// TIA Portal V17 export
// export: Created 2023-03-03T08:59:14.9842508Z, ExportSetting WithDefaults, DisplayName Totally Integrated Automation Portal, DisplayVersion V17 Update 5, DisplayName TIA Portal Openness, DisplayVersion V17 Update 5, DisplayName TIA Portal Version Control Interface, DisplayVersion V17, DisplayName SINAMICS Startdrive Advanced, DisplayVersion V17 SP1, DisplayName SINAMICS DCC, DisplayVersion V17 Update 1, DisplayName SINAMICS Startdrive G130, G150, S120, S150, SINAMICS MV, S210, DisplayVersion V17 SP1, DisplayName SINAMICS Startdrive G110M, G120, G120C, G120D, G120P, G115D, DisplayVersion V17 SP1, DisplayName STEP 7 Professional, DisplayVersion V17 Update 5, DisplayName STEP 7 Safety, DisplayVersion V17, DisplayName WinCC Advanced, DisplayVersion V17 Update 5
FUNCTION "Lubrification" : Void   // FC600, LAD
TITLE = FC Gestione lubrificazione impianto
{ S7_Optimized_Access := 'FALSE' }
AUTHOR : max
FAMILY : Taglio
NAME : FC_LUBRIFICAZIONE
VERSION : 0.1
// stored: AutoNumber false, IsIECCheckEnabled false, SetENOAutomatically false, UDAEnableTagReadback false
   VAR_TEMP   // added for the SCL form of the ladder/FBD networks
      _w1 : Bool;
      _w2 : Bool;
      _w3 : Bool;
      _w4 : Bool;
   END_VAR
BEGIN

REGION Network 1: ****************************** Lubrificazione cesoia *************************************
END_REGION

REGION Network 2: Condizioni per consenso abilitazione
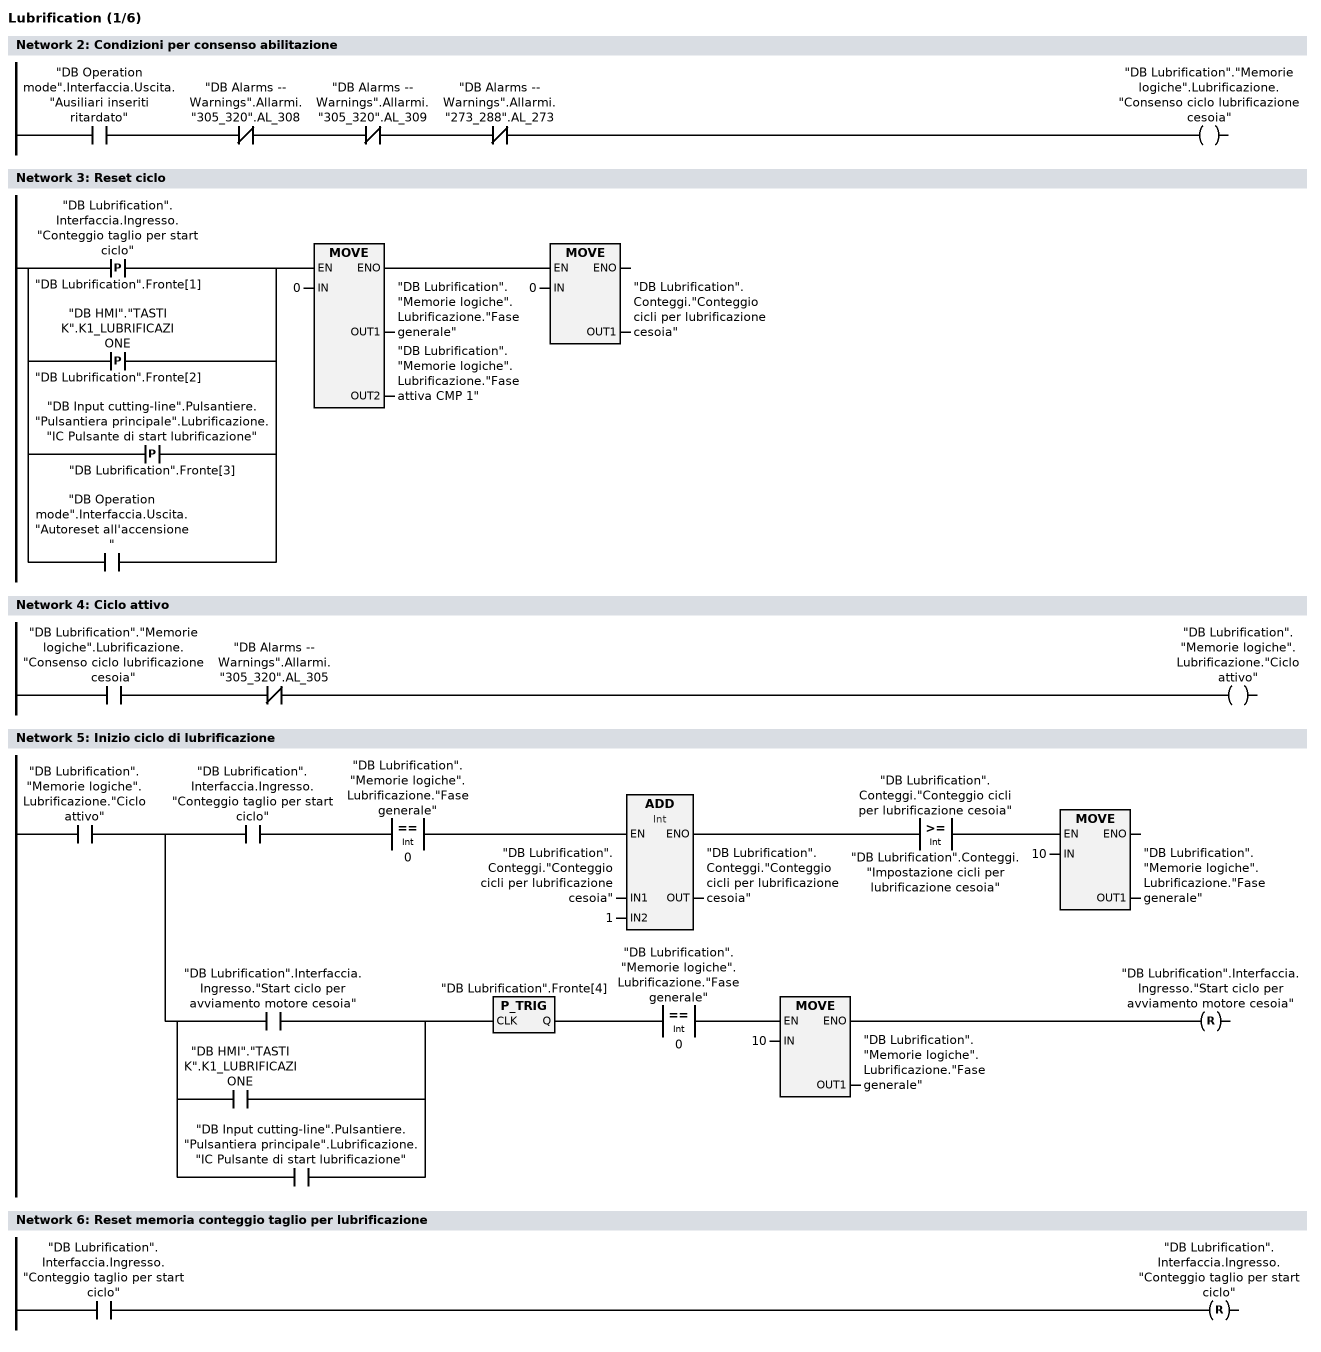
   RUNG wire#powerrail
      Contact( "DB Operation mode".Interfaccia.Uscita."Ausiliari inseriti ritardato" )
      I_Contact( "DB Alarms -- Warnings".Allarmi."305_320".AL_308 )
      I_Contact( "DB Alarms -- Warnings".Allarmi."305_320".AL_309 )
      I_Contact( "DB Alarms -- Warnings".Allarmi."273_288".AL_273 )
      Coil( "DB Lubrification"."Memorie logiche".Lubrificazione."Consenso ciclo lubrificazione cesoia" )
   END_RUNG
   // the same network as SCL:
   "DB Lubrification"."Memorie logiche".Lubrificazione."Consenso ciclo lubrificazione cesoia" := "DB Operation mode".Interfaccia.Uscita."Ausiliari inseriti ritardato" AND NOT "DB Alarms -- Warnings".Allarmi."305_320".AL_308 AND NOT "DB Alarms -- Warnings".Allarmi."305_320".AL_309 AND NOT "DB Alarms -- Warnings".Allarmi."273_288".AL_273;
END_REGION

REGION Network 3: Reset ciclo
   RUNG wire#powerrail
      P_Contact(operand := "DB Lubrification".Interfaccia.Ingresso."Conteggio taglio per start ciclo", bit := "DB Lubrification".Fronte[1])
      wire#w1
      Move(in := 0, out1 => "DB Lubrification"."Memorie logiche".Lubrificazione."Fase generale", out2 => "DB Lubrification"."Memorie logiche".Lubrificazione."Fase attiva CMP 1")
      Move(in := 0, out1 => "DB Lubrification".Conteggi."Conteggio cicli per lubrificazione cesoia")
   END_RUNG
   RUNG wire#powerrail
      P_Contact(operand := "DB HMI"."TASTI K".K1_LUBRIFICAZIONE, bit := "DB Lubrification".Fronte[2])
   END_RUNG wire#w1
   RUNG wire#powerrail
      P_Contact(operand := "DB Input cutting-line".Pulsantiere."Pulsantiera principale".Lubrificazione."IC Pulsante di start lubrificazione", bit := "DB Lubrification".Fronte[3])
   END_RUNG wire#w1
   RUNG wire#powerrail
      Contact( "DB Operation mode".Interfaccia.Uscita."Autoreset all'accensione" )
   END_RUNG wire#w1
   // the same network as SCL:
   #_w1 := "DB Lubrification".Interfaccia.Ingresso."Conteggio taglio per start ciclo" AND NOT "DB Lubrification".Fronte[1];   // rising edge of "DB Lubrification".Interfaccia.Ingresso."Conteggio taglio per start ciclo"
   "DB Lubrification".Fronte[1] := "DB Lubrification".Interfaccia.Ingresso."Conteggio taglio per start ciclo";
   #_w2 := "DB HMI"."TASTI K".K1_LUBRIFICAZIONE AND NOT "DB Lubrification".Fronte[2];   // rising edge of "DB HMI"."TASTI K".K1_LUBRIFICAZIONE
   "DB Lubrification".Fronte[2] := "DB HMI"."TASTI K".K1_LUBRIFICAZIONE;
   #_w3 := "DB Input cutting-line".Pulsantiere."Pulsantiera principale".Lubrificazione."IC Pulsante di start lubrificazione" AND NOT "DB Lubrification".Fronte[3];   // rising edge of "DB Input cutting-line".Pulsantiere."Pulsantiera principale".Lubrificazione."IC Pulsante di start lubrificazione"
   "DB Lubrification".Fronte[3] := "DB Input cutting-line".Pulsantiere."Pulsantiera principale".Lubrificazione."IC Pulsante di start lubrificazione";
   IF #_w1 OR #_w2 OR #_w3 OR "DB Operation mode".Interfaccia.Uscita."Autoreset all'accensione" THEN
       "DB Lubrification"."Memorie logiche".Lubrificazione."Fase generale" := 0;
       "DB Lubrification"."Memorie logiche".Lubrificazione."Fase attiva CMP 1" := 0;
       "DB Lubrification".Conteggi."Conteggio cicli per lubrificazione cesoia" := 0;
   END_IF;
END_REGION

REGION Network 4: Ciclo attivo
   RUNG wire#powerrail
      Contact( "DB Lubrification"."Memorie logiche".Lubrificazione."Consenso ciclo lubrificazione cesoia" )
      I_Contact( "DB Alarms -- Warnings".Allarmi."305_320".AL_305 )
      Coil( "DB Lubrification"."Memorie logiche".Lubrificazione."Ciclo attivo" )
   END_RUNG
   // the same network as SCL:
   "DB Lubrification"."Memorie logiche".Lubrificazione."Ciclo attivo" := "DB Lubrification"."Memorie logiche".Lubrificazione."Consenso ciclo lubrificazione cesoia" AND NOT "DB Alarms -- Warnings".Allarmi."305_320".AL_305;
END_REGION

REGION Network 5: Inizio ciclo di lubrificazione
   RUNG wire#powerrail
      Contact( "DB Lubrification"."Memorie logiche".Lubrificazione."Ciclo attivo" )
      wire#w1
      Contact( "DB Lubrification".Interfaccia.Ingresso."Conteggio taglio per start ciclo" )
      { S7_Templates := "SrcType := Int" } EQ_Contact(in1 := "DB Lubrification"."Memorie logiche".Lubrificazione."Fase generale", in2 := 0)
      { S7_Templates := "SrcType := Int"; S7_GenerateENO := "TRUE" } Add(in1 := "DB Lubrification".Conteggi."Conteggio cicli per lubrificazione cesoia", in2 := 1, out => "DB Lubrification".Conteggi."Conteggio cicli per lubrificazione cesoia")
      { S7_Templates := "SrcType := Int" } GE_Contact(in1 := "DB Lubrification".Conteggi."Conteggio cicli per lubrificazione cesoia", in2 := "DB Lubrification".Conteggi."Impostazione cicli per lubrificazione cesoia")
      Move(in := 10, out1 => "DB Lubrification"."Memorie logiche".Lubrificazione."Fase generale")
   END_RUNG
   RUNG wire#w1
      Contact( "DB Lubrification".Interfaccia.Ingresso."Start ciclo per avviamento motore cesoia" )
      wire#w2
      P_Trig( "DB Lubrification".Fronte[4] )
      { S7_Templates := "SrcType := Int" } EQ_Contact(in1 := "DB Lubrification"."Memorie logiche".Lubrificazione."Fase generale", in2 := 0)
      Move(in := 10, out1 => "DB Lubrification"."Memorie logiche".Lubrificazione."Fase generale")
      R_Coil( "DB Lubrification".Interfaccia.Ingresso."Start ciclo per avviamento motore cesoia" )
   END_RUNG
   RUNG wire#w1
      Contact( "DB HMI"."TASTI K".K1_LUBRIFICAZIONE )
   END_RUNG wire#w2
   RUNG wire#w1
      Contact( "DB Input cutting-line".Pulsantiere."Pulsantiera principale".Lubrificazione."IC Pulsante di start lubrificazione" )
   END_RUNG wire#w2
   // the same network as SCL:
   // ENO of a box is taken as its EN; it also drops when the box reports an error
   #_w1 := "DB Lubrification"."Memorie logiche".Lubrificazione."Ciclo attivo" AND "DB Lubrification".Interfaccia.Ingresso."Conteggio taglio per start ciclo" AND ("DB Lubrification"."Memorie logiche".Lubrificazione."Fase generale" = 0);
   IF #_w1 THEN
       "DB Lubrification".Conteggi."Conteggio cicli per lubrificazione cesoia" := "DB Lubrification".Conteggi."Conteggio cicli per lubrificazione cesoia" + 1;
   END_IF;
   IF #_w1 AND ("DB Lubrification".Conteggi."Conteggio cicli per lubrificazione cesoia" >= "DB Lubrification".Conteggi."Impostazione cicli per lubrificazione cesoia") THEN
       "DB Lubrification"."Memorie logiche".Lubrificazione."Fase generale" := 10;
   END_IF;
   #_w2 := "DB Lubrification"."Memorie logiche".Lubrificazione."Ciclo attivo" AND ("DB Lubrification".Interfaccia.Ingresso."Start ciclo per avviamento motore cesoia" OR "DB HMI"."TASTI K".K1_LUBRIFICAZIONE OR "DB Input cutting-line".Pulsantiere."Pulsantiera principale".Lubrificazione."IC Pulsante di start lubrificazione");
   #_w3 := #_w2 AND NOT "DB Lubrification".Fronte[4];   // rising edge
   "DB Lubrification".Fronte[4] := #_w2;
   #_w4 := #_w3 AND ("DB Lubrification"."Memorie logiche".Lubrificazione."Fase generale" = 0);
   IF #_w4 THEN
       "DB Lubrification"."Memorie logiche".Lubrificazione."Fase generale" := 10;
       "DB Lubrification".Interfaccia.Ingresso."Start ciclo per avviamento motore cesoia" := FALSE;
   END_IF;
END_REGION

REGION Network 6: Reset memoria conteggio taglio per lubrificazione
   RUNG wire#powerrail
      Contact( "DB Lubrification".Interfaccia.Ingresso."Conteggio taglio per start ciclo" )
      R_Coil( "DB Lubrification".Interfaccia.Ingresso."Conteggio taglio per start ciclo" )
   END_RUNG
   // the same network as SCL:
   IF "DB Lubrification".Interfaccia.Ingresso."Conteggio taglio per start ciclo" THEN
       "DB Lubrification".Interfaccia.Ingresso."Conteggio taglio per start ciclo" := FALSE;
   END_IF;
END_REGION

REGION Network 7: Fase10 generale: Verifica stato CMP ad inizio ciclo
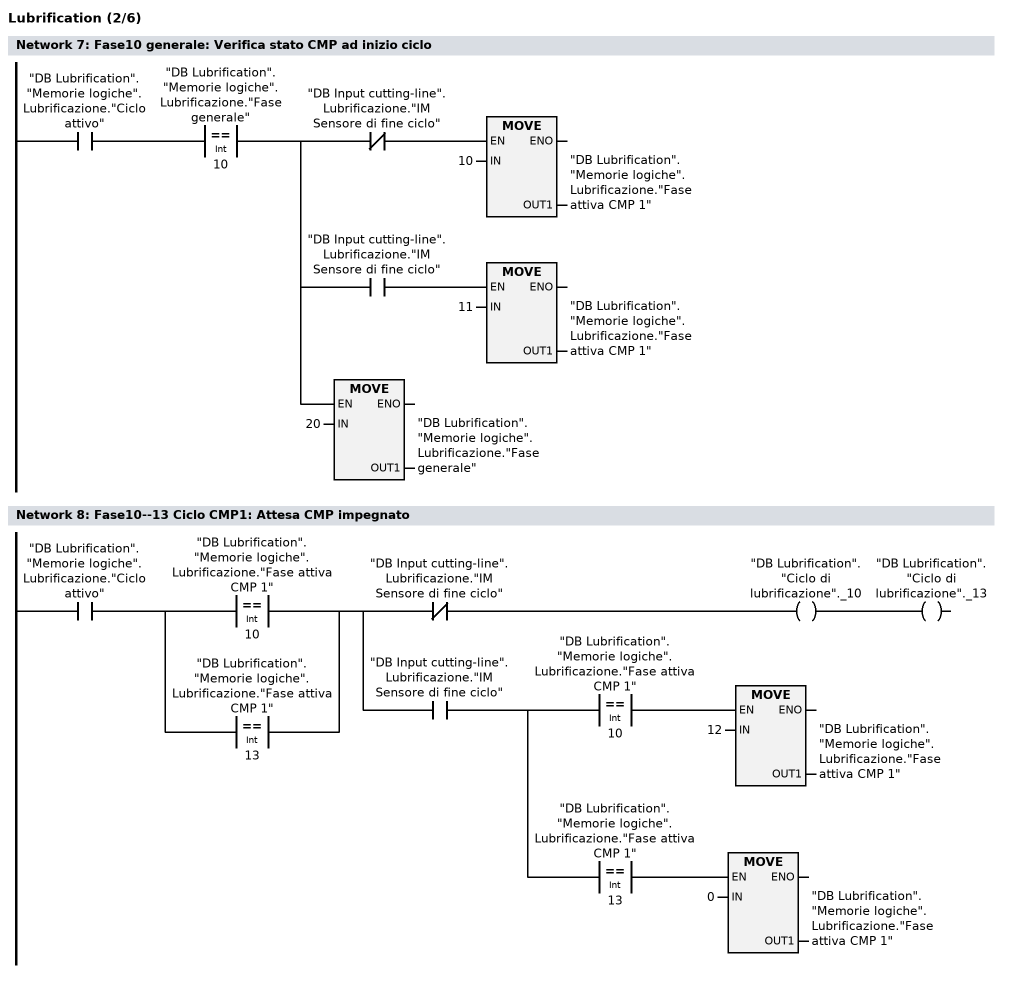
   RUNG wire#powerrail
      Contact( "DB Lubrification"."Memorie logiche".Lubrificazione."Ciclo attivo" )
      { S7_Templates := "SrcType := Int" } EQ_Contact(in1 := "DB Lubrification"."Memorie logiche".Lubrificazione."Fase generale", in2 := 10)
      wire#w1
      I_Contact( "DB Input cutting-line".Lubrificazione."IM Sensore di fine ciclo" )
      Move(in := 10, out1 => "DB Lubrification"."Memorie logiche".Lubrificazione."Fase attiva CMP 1")
   END_RUNG
   RUNG wire#w1
      Contact( "DB Input cutting-line".Lubrificazione."IM Sensore di fine ciclo" )
      Move(in := 11, out1 => "DB Lubrification"."Memorie logiche".Lubrificazione."Fase attiva CMP 1")
   END_RUNG
   RUNG wire#w1
      Move(in := 20, out1 => "DB Lubrification"."Memorie logiche".Lubrificazione."Fase generale")
   END_RUNG
   // the same network as SCL:
   #_w1 := "DB Lubrification"."Memorie logiche".Lubrificazione."Ciclo attivo" AND ("DB Lubrification"."Memorie logiche".Lubrificazione."Fase generale" = 10);
   IF #_w1 AND NOT "DB Input cutting-line".Lubrificazione."IM Sensore di fine ciclo" THEN
       "DB Lubrification"."Memorie logiche".Lubrificazione."Fase attiva CMP 1" := 10;
   END_IF;
   IF #_w1 AND "DB Input cutting-line".Lubrificazione."IM Sensore di fine ciclo" THEN
       "DB Lubrification"."Memorie logiche".Lubrificazione."Fase attiva CMP 1" := 11;
   END_IF;
   IF #_w1 THEN "DB Lubrification"."Memorie logiche".Lubrificazione."Fase generale" := 20; END_IF;
END_REGION

REGION Network 8: Fase10--13 Ciclo CMP1: Attesa CMP impegnato
   RUNG wire#powerrail
      Contact( "DB Lubrification"."Memorie logiche".Lubrificazione."Ciclo attivo" )
      wire#w1
      { S7_Templates := "SrcType := Int" } EQ_Contact(in1 := "DB Lubrification"."Memorie logiche".Lubrificazione."Fase attiva CMP 1", in2 := 10)
      wire#w2
      I_Contact( "DB Input cutting-line".Lubrificazione."IM Sensore di fine ciclo" )
      Coil( "DB Lubrification"."Ciclo di lubrificazione"._10 )
      Coil( "DB Lubrification"."Ciclo di lubrificazione"._13 )
   END_RUNG
   RUNG wire#w1
      { S7_Templates := "SrcType := Int" } EQ_Contact(in1 := "DB Lubrification"."Memorie logiche".Lubrificazione."Fase attiva CMP 1", in2 := 13)
   END_RUNG wire#w2
   RUNG wire#w2
      Contact( "DB Input cutting-line".Lubrificazione."IM Sensore di fine ciclo" )
      wire#w3
      { S7_Templates := "SrcType := Int" } EQ_Contact(in1 := "DB Lubrification"."Memorie logiche".Lubrificazione."Fase attiva CMP 1", in2 := 10)
      Move(in := 12, out1 => "DB Lubrification"."Memorie logiche".Lubrificazione."Fase attiva CMP 1")
   END_RUNG
   RUNG wire#w3
      { S7_Templates := "SrcType := Int" } EQ_Contact(in1 := "DB Lubrification"."Memorie logiche".Lubrificazione."Fase attiva CMP 1", in2 := 13)
      Move(in := 0, out1 => "DB Lubrification"."Memorie logiche".Lubrificazione."Fase attiva CMP 1")
   END_RUNG
   // the same network as SCL:
   #_w1 := "DB Lubrification"."Memorie logiche".Lubrificazione."Ciclo attivo" AND (("DB Lubrification"."Memorie logiche".Lubrificazione."Fase attiva CMP 1" = 10) OR ("DB Lubrification"."Memorie logiche".Lubrificazione."Fase attiva CMP 1" = 13));
   "DB Lubrification"."Ciclo di lubrificazione"._10 := #_w1 AND NOT "DB Input cutting-line".Lubrificazione."IM Sensore di fine ciclo";
   "DB Lubrification"."Ciclo di lubrificazione"._13 := "DB Lubrification"."Ciclo di lubrificazione"._10;
   #_w2 := #_w1 AND "DB Input cutting-line".Lubrificazione."IM Sensore di fine ciclo";
   IF #_w2 AND ("DB Lubrification"."Memorie logiche".Lubrificazione."Fase attiva CMP 1" = 10) THEN
       "DB Lubrification"."Memorie logiche".Lubrificazione."Fase attiva CMP 1" := 12;
   END_IF;
   IF #_w2 AND ("DB Lubrification"."Memorie logiche".Lubrificazione."Fase attiva CMP 1" = 13) THEN
       "DB Lubrification"."Memorie logiche".Lubrificazione."Fase attiva CMP 1" := 0;
   END_IF;
END_REGION

REGION Network 9: Fase11--12 Ciclo CMP1: Attesa CMP dimpegnato
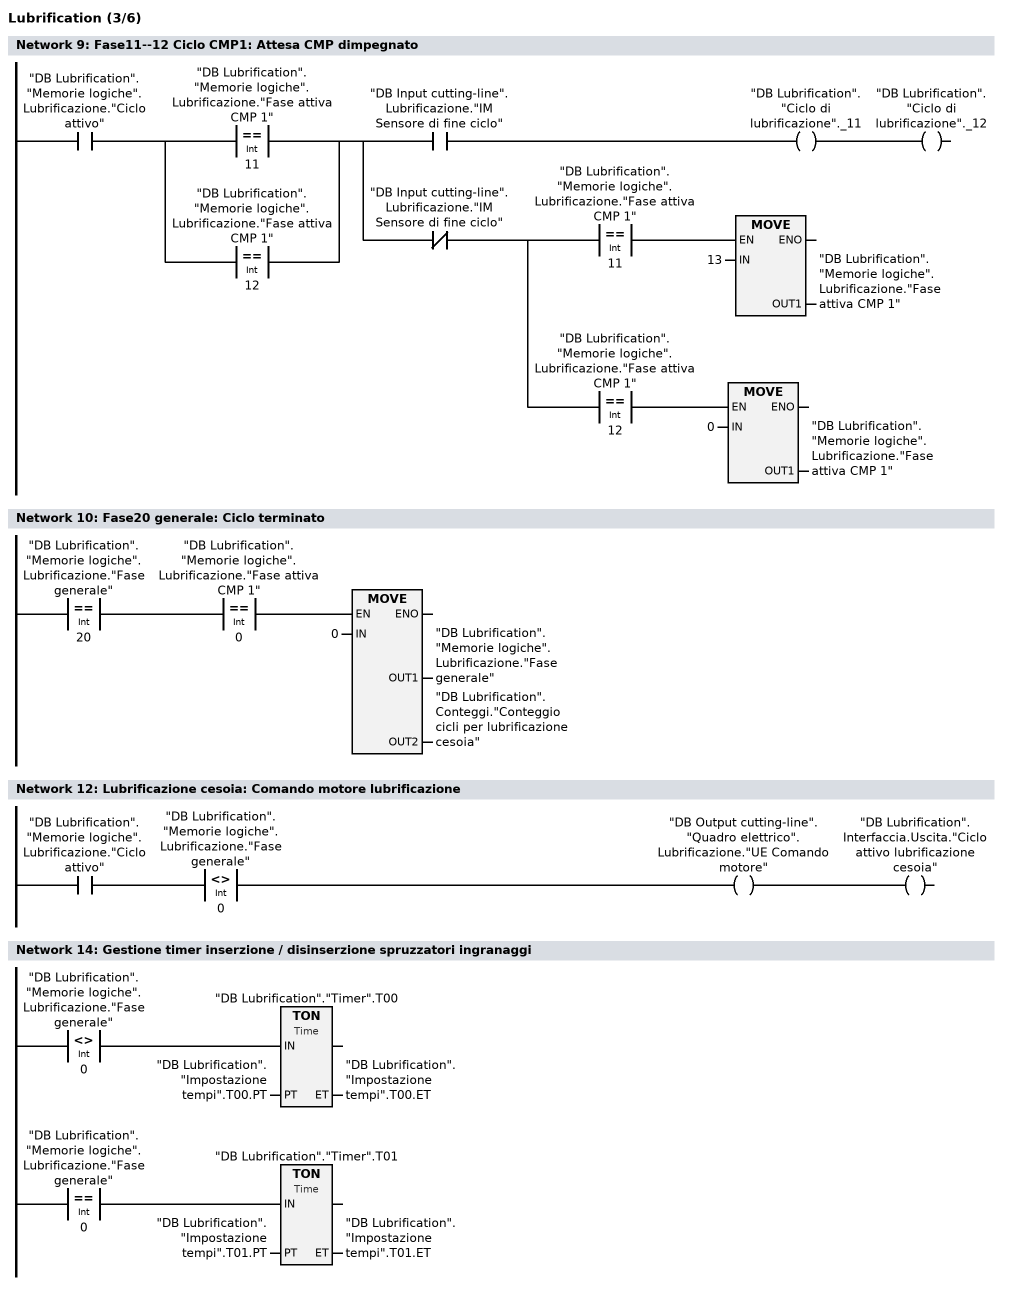
   RUNG wire#powerrail
      Contact( "DB Lubrification"."Memorie logiche".Lubrificazione."Ciclo attivo" )
      wire#w1
      { S7_Templates := "SrcType := Int" } EQ_Contact(in1 := "DB Lubrification"."Memorie logiche".Lubrificazione."Fase attiva CMP 1", in2 := 11)
      wire#w2
      Contact( "DB Input cutting-line".Lubrificazione."IM Sensore di fine ciclo" )
      Coil( "DB Lubrification"."Ciclo di lubrificazione"._11 )
      Coil( "DB Lubrification"."Ciclo di lubrificazione"._12 )
   END_RUNG
   RUNG wire#w1
      { S7_Templates := "SrcType := Int" } EQ_Contact(in1 := "DB Lubrification"."Memorie logiche".Lubrificazione."Fase attiva CMP 1", in2 := 12)
   END_RUNG wire#w2
   RUNG wire#w2
      I_Contact( "DB Input cutting-line".Lubrificazione."IM Sensore di fine ciclo" )
      wire#w3
      { S7_Templates := "SrcType := Int" } EQ_Contact(in1 := "DB Lubrification"."Memorie logiche".Lubrificazione."Fase attiva CMP 1", in2 := 11)
      Move(in := 13, out1 => "DB Lubrification"."Memorie logiche".Lubrificazione."Fase attiva CMP 1")
   END_RUNG
   RUNG wire#w3
      { S7_Templates := "SrcType := Int" } EQ_Contact(in1 := "DB Lubrification"."Memorie logiche".Lubrificazione."Fase attiva CMP 1", in2 := 12)
      Move(in := 0, out1 => "DB Lubrification"."Memorie logiche".Lubrificazione."Fase attiva CMP 1")
   END_RUNG
   // the same network as SCL:
   #_w1 := "DB Lubrification"."Memorie logiche".Lubrificazione."Ciclo attivo" AND (("DB Lubrification"."Memorie logiche".Lubrificazione."Fase attiva CMP 1" = 11) OR ("DB Lubrification"."Memorie logiche".Lubrificazione."Fase attiva CMP 1" = 12));
   "DB Lubrification"."Ciclo di lubrificazione"._11 := #_w1 AND "DB Input cutting-line".Lubrificazione."IM Sensore di fine ciclo";
   "DB Lubrification"."Ciclo di lubrificazione"._12 := "DB Lubrification"."Ciclo di lubrificazione"._11;
   #_w2 := #_w1 AND NOT "DB Input cutting-line".Lubrificazione."IM Sensore di fine ciclo";
   IF #_w2 AND ("DB Lubrification"."Memorie logiche".Lubrificazione."Fase attiva CMP 1" = 11) THEN
       "DB Lubrification"."Memorie logiche".Lubrificazione."Fase attiva CMP 1" := 13;
   END_IF;
   IF #_w2 AND ("DB Lubrification"."Memorie logiche".Lubrificazione."Fase attiva CMP 1" = 12) THEN
       "DB Lubrification"."Memorie logiche".Lubrificazione."Fase attiva CMP 1" := 0;
   END_IF;
END_REGION

REGION Network 10: Fase20 generale: Ciclo terminato
   RUNG wire#powerrail
      { S7_Templates := "SrcType := Int" } EQ_Contact(in1 := "DB Lubrification"."Memorie logiche".Lubrificazione."Fase generale", in2 := 20)
      { S7_Templates := "SrcType := Int" } EQ_Contact(in1 := "DB Lubrification"."Memorie logiche".Lubrificazione."Fase attiva CMP 1", in2 := 0)
      Move(in := 0, out1 => "DB Lubrification"."Memorie logiche".Lubrificazione."Fase generale", out2 => "DB Lubrification".Conteggi."Conteggio cicli per lubrificazione cesoia")
   END_RUNG
   // the same network as SCL:
   IF ("DB Lubrification"."Memorie logiche".Lubrificazione."Fase generale" = 20) AND ("DB Lubrification"."Memorie logiche".Lubrificazione."Fase attiva CMP 1" = 0) THEN
       "DB Lubrification"."Memorie logiche".Lubrificazione."Fase generale" := 0;
       "DB Lubrification".Conteggi."Conteggio cicli per lubrificazione cesoia" := 0;
   END_IF;
END_REGION

REGION Network 11: Dummy
END_REGION

REGION Network 12: Lubrificazione cesoia: Comando motore lubrificazione
   RUNG wire#powerrail
      Contact( "DB Lubrification"."Memorie logiche".Lubrificazione."Ciclo attivo" )
      { S7_Templates := "SrcType := Int" } NE_Contact(in1 := "DB Lubrification"."Memorie logiche".Lubrificazione."Fase generale", in2 := 0)
      Coil( "DB Output cutting-line"."Quadro elettrico".Lubrificazione."UE Comando motore" )
      Coil( "DB Lubrification".Interfaccia.Uscita."Ciclo attivo lubrificazione cesoia" )
   END_RUNG
   // the same network as SCL:
   "DB Output cutting-line"."Quadro elettrico".Lubrificazione."UE Comando motore" := "DB Lubrification"."Memorie logiche".Lubrificazione."Ciclo attivo" AND ("DB Lubrification"."Memorie logiche".Lubrificazione."Fase generale" <> 0);
   "DB Lubrification".Interfaccia.Uscita."Ciclo attivo lubrificazione cesoia" := "DB Output cutting-line"."Quadro elettrico".Lubrificazione."UE Comando motore";
END_REGION

REGION Network 13: Dummy
END_REGION

REGION Network 14: Gestione timer inserzione / disinserzione spruzzatori ingranaggi
   RUNG wire#powerrail
      { S7_Templates := "SrcType := Int" } NE_Contact(in1 := "DB Lubrification"."Memorie logiche".Lubrificazione."Fase generale", in2 := 0)
      { S7_Templates := "time_type := Time" } "DB Lubrification"."Timer".T00.TON(pt := "DB Lubrification"."Impostazione tempi".T00.PT, et => "DB Lubrification"."Impostazione tempi".T00.ET)
   END_RUNG
   RUNG wire#powerrail
      { S7_Templates := "SrcType := Int" } EQ_Contact(in1 := "DB Lubrification"."Memorie logiche".Lubrificazione."Fase generale", in2 := 0)
      { S7_Templates := "time_type := Time" } "DB Lubrification"."Timer".T01.TON(pt := "DB Lubrification"."Impostazione tempi".T01.PT, et => "DB Lubrification"."Impostazione tempi".T01.ET)
   END_RUNG
   // the same network as SCL:
   "DB Lubrification"."Timer".T00.TON(IN := "DB Lubrification"."Memorie logiche".Lubrificazione."Fase generale" <> 0,
                           PT := "DB Lubrification"."Impostazione tempi".T00.PT,
                           ET => "DB Lubrification"."Impostazione tempi".T00.ET);
   "DB Lubrification"."Timer".T01.TON(IN := "DB Lubrification"."Memorie logiche".Lubrificazione."Fase generale" = 0,
                           PT := "DB Lubrification"."Impostazione tempi".T01.PT,
                           ET => "DB Lubrification"."Impostazione tempi".T01.ET);
END_REGION

REGION Network 15: Lubrificazione cesoia: Comando spruzzatori ingranaggi
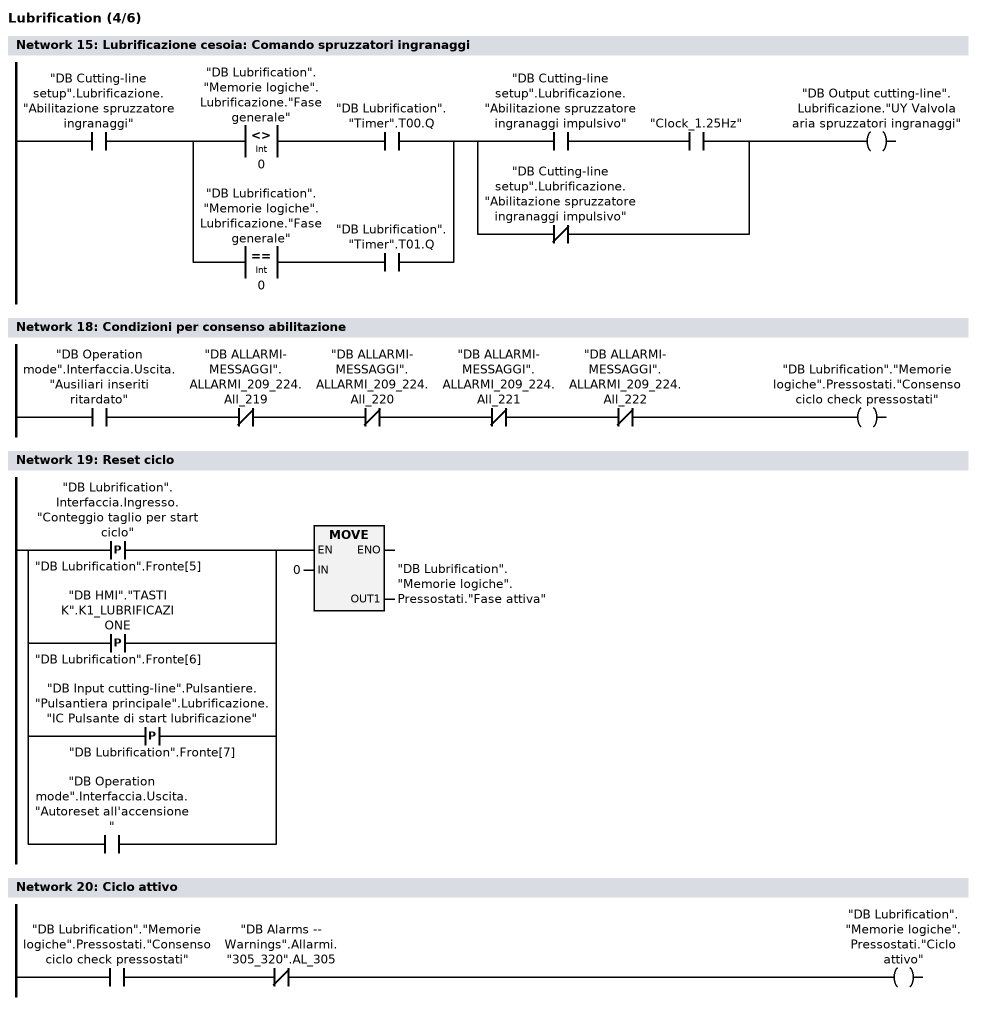
   RUNG wire#powerrail
      Contact( "DB Cutting-line setup".Lubrificazione."Abilitazione spruzzatore ingranaggi" )
      wire#w1
      { S7_Templates := "SrcType := Int" } NE_Contact(in1 := "DB Lubrification"."Memorie logiche".Lubrificazione."Fase generale", in2 := 0)
      Contact( "DB Lubrification"."Timer".T00.Q )
      wire#w2
      Contact( "DB Cutting-line setup".Lubrificazione."Abilitazione spruzzatore ingranaggi impulsivo" )
      Contact( "Clock_1.25Hz" )
      wire#w3
      Coil( "DB Output cutting-line".Lubrificazione."UY Valvola aria spruzzatori ingranaggi" )
   END_RUNG
   RUNG wire#w1
      { S7_Templates := "SrcType := Int" } EQ_Contact(in1 := "DB Lubrification"."Memorie logiche".Lubrificazione."Fase generale", in2 := 0)
      Contact( "DB Lubrification"."Timer".T01.Q )
   END_RUNG wire#w2
   RUNG wire#w2
      I_Contact( "DB Cutting-line setup".Lubrificazione."Abilitazione spruzzatore ingranaggi impulsivo" )
   END_RUNG wire#w3
   // the same network as SCL:
   "DB Output cutting-line".Lubrificazione."UY Valvola aria spruzzatori ingranaggi" := "DB Cutting-line setup".Lubrificazione."Abilitazione spruzzatore ingranaggi" AND ((("DB Lubrification"."Memorie logiche".Lubrificazione."Fase generale" <> 0) AND "DB Lubrification"."Timer".T00.Q) OR (("DB Lubrification"."Memorie logiche".Lubrificazione."Fase generale" = 0) AND "DB Lubrification"."Timer".T01.Q)) AND (("DB Cutting-line setup".Lubrificazione."Abilitazione spruzzatore ingranaggi impulsivo" AND "Clock_1.25Hz") OR NOT "DB Cutting-line setup".Lubrificazione."Abilitazione spruzzatore ingranaggi impulsivo");
END_REGION

REGION Network 16: Dummy
END_REGION

REGION Network 17: ******************************* Check pressostati **************************************
END_REGION

REGION Network 18: Condizioni per consenso abilitazione
   RUNG wire#powerrail
      Contact( "DB Operation mode".Interfaccia.Uscita."Ausiliari inseriti ritardato" )
      I_Contact( "DB ALLARMI-MESSAGGI".ALLARMI_209_224.All_219 )
      I_Contact( "DB ALLARMI-MESSAGGI".ALLARMI_209_224.All_220 )
      I_Contact( "DB ALLARMI-MESSAGGI".ALLARMI_209_224.All_221 )
      I_Contact( "DB ALLARMI-MESSAGGI".ALLARMI_209_224.All_222 )
      Coil( "DB Lubrification"."Memorie logiche".Pressostati."Consenso ciclo check pressostati" )
   END_RUNG
   // the same network as SCL:
   "DB Lubrification"."Memorie logiche".Pressostati."Consenso ciclo check pressostati" := "DB Operation mode".Interfaccia.Uscita."Ausiliari inseriti ritardato" AND NOT "DB ALLARMI-MESSAGGI".ALLARMI_209_224.All_219 AND NOT "DB ALLARMI-MESSAGGI".ALLARMI_209_224.All_220 AND NOT "DB ALLARMI-MESSAGGI".ALLARMI_209_224.All_221 AND NOT "DB ALLARMI-MESSAGGI".ALLARMI_209_224.All_222;
END_REGION

REGION Network 19: Reset ciclo
   RUNG wire#powerrail
      P_Contact(operand := "DB Lubrification".Interfaccia.Ingresso."Conteggio taglio per start ciclo", bit := "DB Lubrification".Fronte[5])
      wire#w1
      Move(in := 0, out1 => "DB Lubrification"."Memorie logiche".Pressostati."Fase attiva")
   END_RUNG
   RUNG wire#powerrail
      P_Contact(operand := "DB HMI"."TASTI K".K1_LUBRIFICAZIONE, bit := "DB Lubrification".Fronte[6])
   END_RUNG wire#w1
   RUNG wire#powerrail
      P_Contact(operand := "DB Input cutting-line".Pulsantiere."Pulsantiera principale".Lubrificazione."IC Pulsante di start lubrificazione", bit := "DB Lubrification".Fronte[7])
   END_RUNG wire#w1
   RUNG wire#powerrail
      Contact( "DB Operation mode".Interfaccia.Uscita."Autoreset all'accensione" )
   END_RUNG wire#w1
   // the same network as SCL:
   #_w1 := "DB Lubrification".Interfaccia.Ingresso."Conteggio taglio per start ciclo" AND NOT "DB Lubrification".Fronte[5];   // rising edge of "DB Lubrification".Interfaccia.Ingresso."Conteggio taglio per start ciclo"
   "DB Lubrification".Fronte[5] := "DB Lubrification".Interfaccia.Ingresso."Conteggio taglio per start ciclo";
   #_w2 := "DB HMI"."TASTI K".K1_LUBRIFICAZIONE AND NOT "DB Lubrification".Fronte[6];   // rising edge of "DB HMI"."TASTI K".K1_LUBRIFICAZIONE
   "DB Lubrification".Fronte[6] := "DB HMI"."TASTI K".K1_LUBRIFICAZIONE;
   #_w3 := "DB Input cutting-line".Pulsantiere."Pulsantiera principale".Lubrificazione."IC Pulsante di start lubrificazione" AND NOT "DB Lubrification".Fronte[7];   // rising edge of "DB Input cutting-line".Pulsantiere."Pulsantiera principale".Lubrificazione."IC Pulsante di start lubrificazione"
   "DB Lubrification".Fronte[7] := "DB Input cutting-line".Pulsantiere."Pulsantiera principale".Lubrificazione."IC Pulsante di start lubrificazione";
   IF #_w1 OR #_w2 OR #_w3 OR "DB Operation mode".Interfaccia.Uscita."Autoreset all'accensione" THEN
       "DB Lubrification"."Memorie logiche".Pressostati."Fase attiva" := 0;
   END_IF;
END_REGION

REGION Network 20: Ciclo attivo
   RUNG wire#powerrail
      Contact( "DB Lubrification"."Memorie logiche".Pressostati."Consenso ciclo check pressostati" )
      I_Contact( "DB Alarms -- Warnings".Allarmi."305_320".AL_305 )
      Coil( "DB Lubrification"."Memorie logiche".Pressostati."Ciclo attivo" )
   END_RUNG
   // the same network as SCL:
   "DB Lubrification"."Memorie logiche".Pressostati."Ciclo attivo" := "DB Lubrification"."Memorie logiche".Pressostati."Consenso ciclo check pressostati" AND NOT "DB Alarms -- Warnings".Allarmi."305_320".AL_305;
END_REGION

REGION Network 21: Inizio ciclo check pressostati
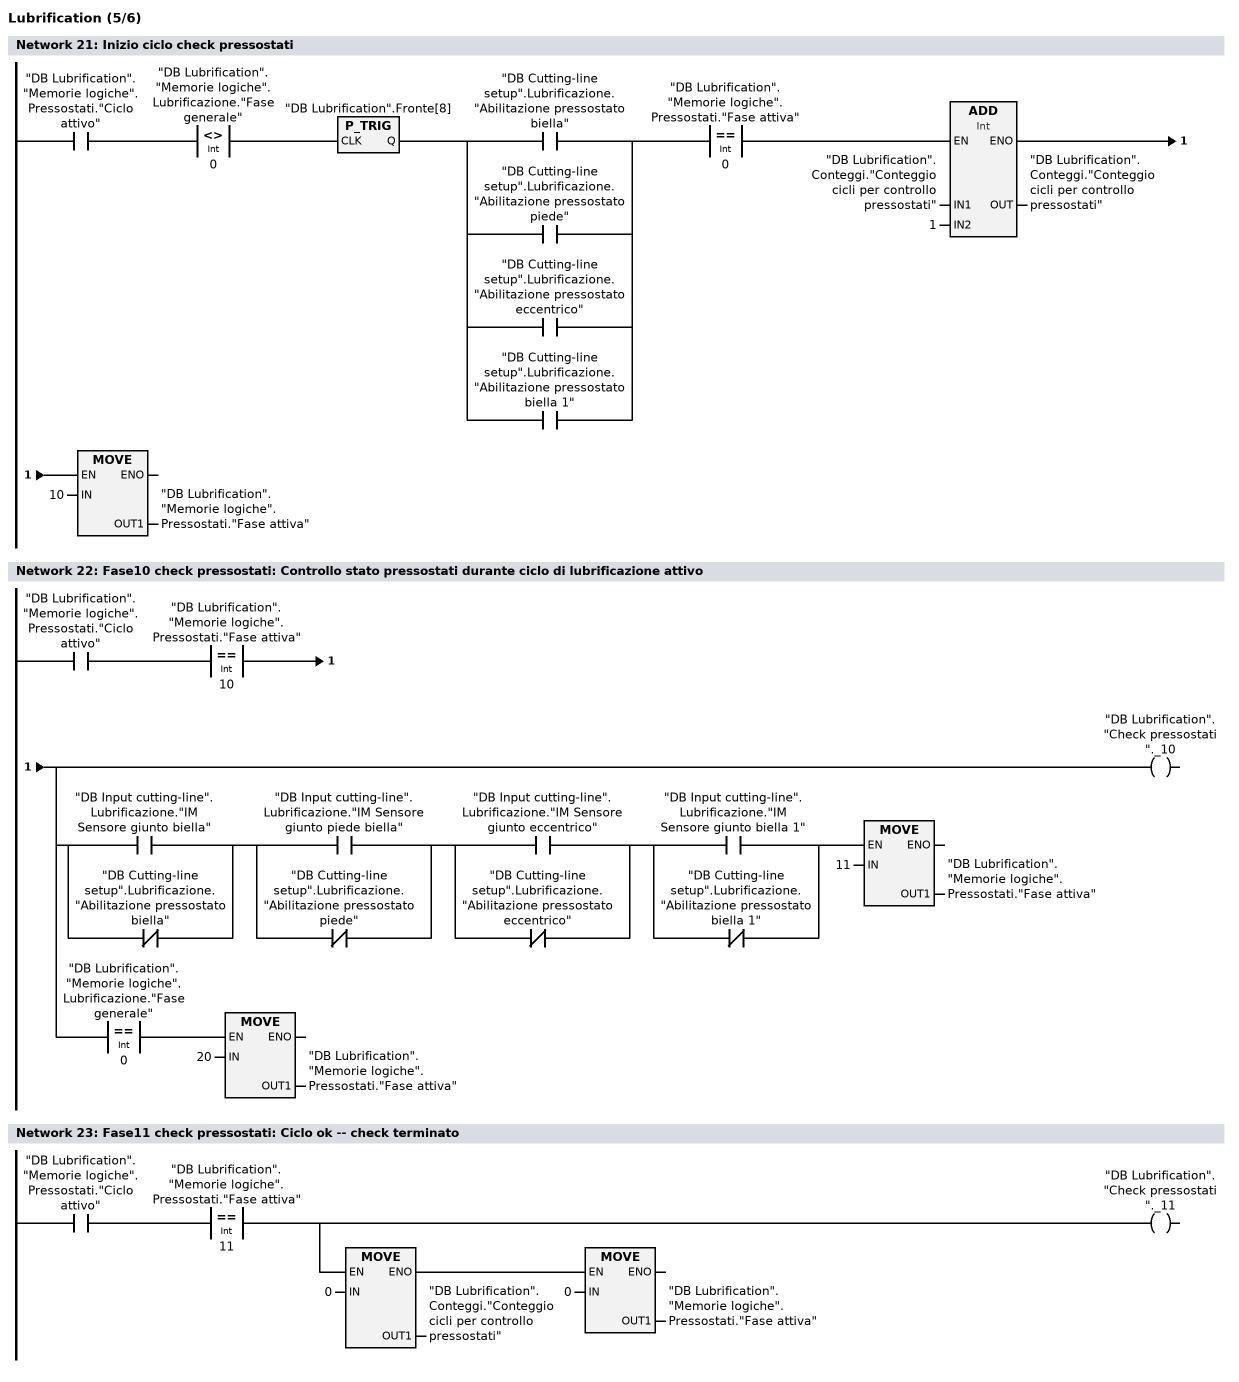
   RUNG wire#powerrail
      Contact( "DB Lubrification"."Memorie logiche".Pressostati."Ciclo attivo" )
      { S7_Templates := "SrcType := Int" } NE_Contact(in1 := "DB Lubrification"."Memorie logiche".Lubrificazione."Fase generale", in2 := 0)
      P_Trig( "DB Lubrification".Fronte[8] )
      wire#w1
      Contact( "DB Cutting-line setup".Lubrificazione."Abilitazione pressostato biella" )
      wire#w2
      { S7_Templates := "SrcType := Int" } EQ_Contact(in1 := "DB Lubrification"."Memorie logiche".Pressostati."Fase attiva", in2 := 0)
      { S7_Templates := "SrcType := Int"; S7_GenerateENO := "TRUE" } Add(in1 := "DB Lubrification".Conteggi."Conteggio cicli per controllo pressostati", in2 := 1, out => "DB Lubrification".Conteggi."Conteggio cicli per controllo pressostati")
      Move(in := 10, out1 => "DB Lubrification"."Memorie logiche".Pressostati."Fase attiva")
   END_RUNG
   RUNG wire#w1
      Contact( "DB Cutting-line setup".Lubrificazione."Abilitazione pressostato piede" )
   END_RUNG wire#w2
   RUNG wire#w1
      Contact( "DB Cutting-line setup".Lubrificazione."Abilitazione pressostato eccentrico" )
   END_RUNG wire#w2
   RUNG wire#w1
      Contact( "DB Cutting-line setup".Lubrificazione."Abilitazione pressostato biella 1" )
   END_RUNG wire#w2
   // the same network as SCL:
   // ENO of a box is taken as its EN; it also drops when the box reports an error
   #_w1 := "DB Lubrification"."Memorie logiche".Pressostati."Ciclo attivo" AND ("DB Lubrification"."Memorie logiche".Lubrificazione."Fase generale" <> 0);
   #_w2 := #_w1 AND NOT "DB Lubrification".Fronte[8];   // rising edge
   "DB Lubrification".Fronte[8] := #_w1;
   IF #_w2 AND ("DB Cutting-line setup".Lubrificazione."Abilitazione pressostato biella" OR "DB Cutting-line setup".Lubrificazione."Abilitazione pressostato piede" OR "DB Cutting-line setup".Lubrificazione."Abilitazione pressostato eccentrico" OR "DB Cutting-line setup".Lubrificazione."Abilitazione pressostato biella 1") AND ("DB Lubrification"."Memorie logiche".Pressostati."Fase attiva" = 0) THEN
       "DB Lubrification".Conteggi."Conteggio cicli per controllo pressostati" := "DB Lubrification".Conteggi."Conteggio cicli per controllo pressostati" + 1;
       "DB Lubrification"."Memorie logiche".Pressostati."Fase attiva" := 10;
   END_IF;
END_REGION

REGION Network 22: Fase10 check pressostati: Controllo stato pressostati durante ciclo di lubrificazione attivo
   RUNG wire#powerrail
      Contact( "DB Lubrification"."Memorie logiche".Pressostati."Ciclo attivo" )
      { S7_Templates := "SrcType := Int" } EQ_Contact(in1 := "DB Lubrification"."Memorie logiche".Pressostati."Fase attiva", in2 := 10)
      wire#w1
      Coil( "DB Lubrification"."Check pressostati"._10 )
   END_RUNG
   RUNG wire#w1
      Contact( "DB Input cutting-line".Lubrificazione."IM Sensore giunto biella" )
      wire#w2
      Contact( "DB Input cutting-line".Lubrificazione."IM Sensore giunto piede biella" )
      wire#w3
      Contact( "DB Input cutting-line".Lubrificazione."IM Sensore giunto eccentrico" )
      wire#w4
      Contact( "DB Input cutting-line".Lubrificazione."IM Sensore giunto biella 1" )
      wire#w5
      Move(in := 11, out1 => "DB Lubrification"."Memorie logiche".Pressostati."Fase attiva")
   END_RUNG
   RUNG wire#w1
      I_Contact( "DB Cutting-line setup".Lubrificazione."Abilitazione pressostato biella" )
   END_RUNG wire#w2
   RUNG wire#w2
      I_Contact( "DB Cutting-line setup".Lubrificazione."Abilitazione pressostato piede" )
   END_RUNG wire#w3
   RUNG wire#w3
      I_Contact( "DB Cutting-line setup".Lubrificazione."Abilitazione pressostato eccentrico" )
   END_RUNG wire#w4
   RUNG wire#w4
      I_Contact( "DB Cutting-line setup".Lubrificazione."Abilitazione pressostato biella 1" )
   END_RUNG wire#w5
   RUNG wire#w1
      { S7_Templates := "SrcType := Int" } EQ_Contact(in1 := "DB Lubrification"."Memorie logiche".Lubrificazione."Fase generale", in2 := 0)
      Move(in := 20, out1 => "DB Lubrification"."Memorie logiche".Pressostati."Fase attiva")
   END_RUNG
   // the same network as SCL:
   "DB Lubrification"."Check pressostati"._10 := "DB Lubrification"."Memorie logiche".Pressostati."Ciclo attivo" AND ("DB Lubrification"."Memorie logiche".Pressostati."Fase attiva" = 10);
   IF "DB Lubrification"."Check pressostati"._10 AND ("DB Input cutting-line".Lubrificazione."IM Sensore giunto biella" OR NOT "DB Cutting-line setup".Lubrificazione."Abilitazione pressostato biella") AND ("DB Input cutting-line".Lubrificazione."IM Sensore giunto piede biella" OR NOT "DB Cutting-line setup".Lubrificazione."Abilitazione pressostato piede") AND ("DB Input cutting-line".Lubrificazione."IM Sensore giunto eccentrico" OR NOT "DB Cutting-line setup".Lubrificazione."Abilitazione pressostato eccentrico") AND ("DB Input cutting-line".Lubrificazione."IM Sensore giunto biella 1" OR NOT "DB Cutting-line setup".Lubrificazione."Abilitazione pressostato biella 1") THEN
       "DB Lubrification"."Memorie logiche".Pressostati."Fase attiva" := 11;
   END_IF;
   IF "DB Lubrification"."Check pressostati"._10 AND ("DB Lubrification"."Memorie logiche".Lubrificazione."Fase generale" = 0) THEN
       "DB Lubrification"."Memorie logiche".Pressostati."Fase attiva" := 20;
   END_IF;
END_REGION

REGION Network 23: Fase11 check pressostati: Ciclo ok -- check terminato
   RUNG wire#powerrail
      Contact( "DB Lubrification"."Memorie logiche".Pressostati."Ciclo attivo" )
      { S7_Templates := "SrcType := Int" } EQ_Contact(in1 := "DB Lubrification"."Memorie logiche".Pressostati."Fase attiva", in2 := 11)
      wire#w1
      Coil( "DB Lubrification"."Check pressostati"._11 )
   END_RUNG
   RUNG wire#w1
      { S7_GenerateENO := "TRUE" } Move(in := 0, out1 => "DB Lubrification".Conteggi."Conteggio cicli per controllo pressostati")
      Move(in := 0, out1 => "DB Lubrification"."Memorie logiche".Pressostati."Fase attiva")
   END_RUNG
   // the same network as SCL:
   // ENO of a box is taken as its EN; it also drops when the box reports an error
   "DB Lubrification"."Check pressostati"._11 := "DB Lubrification"."Memorie logiche".Pressostati."Ciclo attivo" AND ("DB Lubrification"."Memorie logiche".Pressostati."Fase attiva" = 11);
   IF "DB Lubrification"."Check pressostati"._11 THEN
       "DB Lubrification".Conteggi."Conteggio cicli per controllo pressostati" := 0;
       "DB Lubrification"."Memorie logiche".Pressostati."Fase attiva" := 0;
   END_IF;
END_REGION

REGION Network 24: Fase20 check pressostati: Ciclo non ok -- generazione allarmi pressostati se conteggio terminato
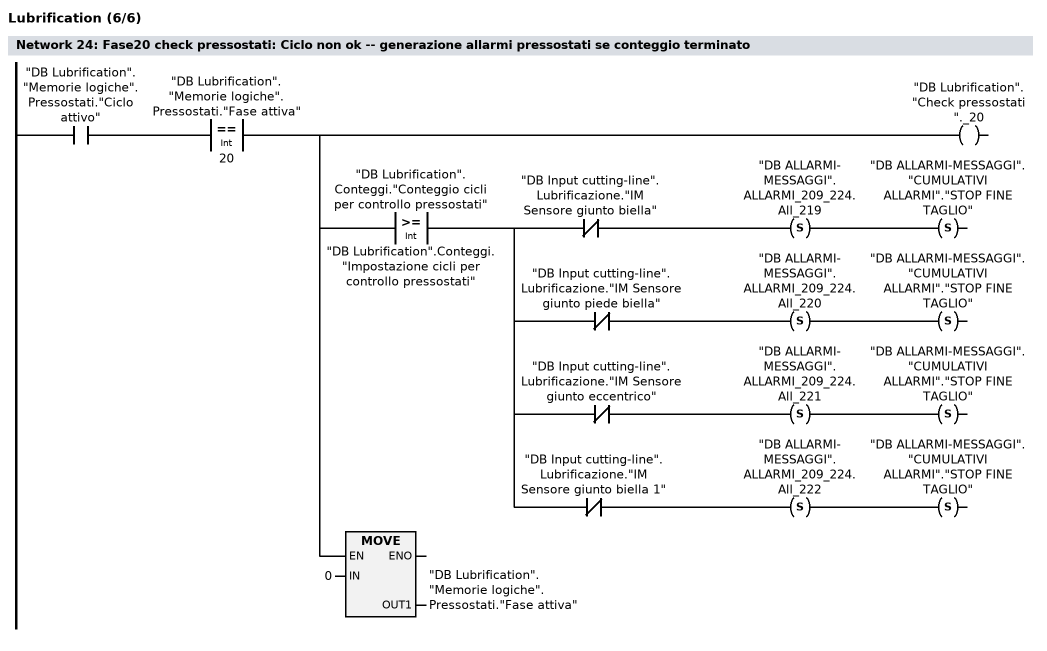
   RUNG wire#powerrail
      Contact( "DB Lubrification"."Memorie logiche".Pressostati."Ciclo attivo" )
      { S7_Templates := "SrcType := Int" } EQ_Contact(in1 := "DB Lubrification"."Memorie logiche".Pressostati."Fase attiva", in2 := 20)
      wire#w1
      Coil( "DB Lubrification"."Check pressostati"._20 )
   END_RUNG
   RUNG wire#w1
      { S7_Templates := "SrcType := Int" } GE_Contact(in1 := "DB Lubrification".Conteggi."Conteggio cicli per controllo pressostati", in2 := "DB Lubrification".Conteggi."Impostazione cicli per controllo pressostati")
      wire#w2
      I_Contact( "DB Input cutting-line".Lubrificazione."IM Sensore giunto biella" )
      S_Coil( "DB ALLARMI-MESSAGGI".ALLARMI_209_224.All_219 )
      S_Coil( "DB ALLARMI-MESSAGGI"."CUMULATIVI ALLARMI"."STOP FINE TAGLIO" )
   END_RUNG
   RUNG wire#w2
      I_Contact( "DB Input cutting-line".Lubrificazione."IM Sensore giunto piede biella" )
      S_Coil( "DB ALLARMI-MESSAGGI".ALLARMI_209_224.All_220 )
      S_Coil( "DB ALLARMI-MESSAGGI"."CUMULATIVI ALLARMI"."STOP FINE TAGLIO" )
   END_RUNG
   RUNG wire#w2
      I_Contact( "DB Input cutting-line".Lubrificazione."IM Sensore giunto eccentrico" )
      S_Coil( "DB ALLARMI-MESSAGGI".ALLARMI_209_224.All_221 )
      S_Coil( "DB ALLARMI-MESSAGGI"."CUMULATIVI ALLARMI"."STOP FINE TAGLIO" )
   END_RUNG
   RUNG wire#w2
      I_Contact( "DB Input cutting-line".Lubrificazione."IM Sensore giunto biella 1" )
      S_Coil( "DB ALLARMI-MESSAGGI".ALLARMI_209_224.All_222 )
      S_Coil( "DB ALLARMI-MESSAGGI"."CUMULATIVI ALLARMI"."STOP FINE TAGLIO" )
   END_RUNG
   RUNG wire#w1
      Move(in := 0, out1 => "DB Lubrification"."Memorie logiche".Pressostati."Fase attiva")
   END_RUNG
   // the same network as SCL:
   "DB Lubrification"."Check pressostati"._20 := "DB Lubrification"."Memorie logiche".Pressostati."Ciclo attivo" AND ("DB Lubrification"."Memorie logiche".Pressostati."Fase attiva" = 20);
   #_w1 := "DB Lubrification"."Check pressostati"._20 AND ("DB Lubrification".Conteggi."Conteggio cicli per controllo pressostati" >= "DB Lubrification".Conteggi."Impostazione cicli per controllo pressostati");
   IF #_w1 AND NOT "DB Input cutting-line".Lubrificazione."IM Sensore giunto biella" THEN
       "DB ALLARMI-MESSAGGI".ALLARMI_209_224.All_219 := TRUE;
       "DB ALLARMI-MESSAGGI"."CUMULATIVI ALLARMI"."STOP FINE TAGLIO" := TRUE;
   END_IF;
   IF #_w1 AND NOT "DB Input cutting-line".Lubrificazione."IM Sensore giunto piede biella" THEN
       "DB ALLARMI-MESSAGGI".ALLARMI_209_224.All_220 := TRUE;
       "DB ALLARMI-MESSAGGI"."CUMULATIVI ALLARMI"."STOP FINE TAGLIO" := TRUE;
   END_IF;
   IF #_w1 AND NOT "DB Input cutting-line".Lubrificazione."IM Sensore giunto eccentrico" THEN
       "DB ALLARMI-MESSAGGI".ALLARMI_209_224.All_221 := TRUE;
       "DB ALLARMI-MESSAGGI"."CUMULATIVI ALLARMI"."STOP FINE TAGLIO" := TRUE;
   END_IF;
   IF #_w1 AND NOT "DB Input cutting-line".Lubrificazione."IM Sensore giunto biella 1" THEN
       "DB ALLARMI-MESSAGGI".ALLARMI_209_224.All_222 := TRUE;
       "DB ALLARMI-MESSAGGI"."CUMULATIVI ALLARMI"."STOP FINE TAGLIO" := TRUE;
   END_IF;
   IF "DB Lubrification"."Check pressostati"._20 THEN
       "DB Lubrification"."Memorie logiche".Pressostati."Fase attiva" := 0;
   END_IF;
END_REGION

REGION Network 25: Dummy
END_REGION
END_FUNCTION
